// TIA Portal V17 export
// export: Created 2025-08-05T09:36:01.5993523Z, ExportSetting WithDefaults, DisplayName Totally Integrated Automation Portal, DisplayVersion V17, DisplayName TIA Portal Openness, DisplayVersion V17, DisplayName TIA Portal Version Control Interface, DisplayVersion V17, DisplayName SINAMICS Startdrive Advanced, DisplayVersion V17, DisplayName SINAMICS Startdrive G130, G150, S120, S150, SINAMICS MV, S210, DisplayVersion V17, DisplayName SINAMICS Startdrive G110M, G120, G120C, G120D, G120P, G115D, DisplayVersion V17, DisplayName STEP 7 Professional, DisplayVersion V17, DisplayName STEP 7 Safety, DisplayVersion V17, DisplayName WinCC Advanced, DisplayVersion V17
TYPE "API_Outputs"
// stored: IsFailsafeCompliant false
   STRUCT
      Job_Comp_Ack : Bool;   // Acknowledge the Job Complete Signal has been Received
      Tx : DInt;   // Transmission Counter
      Job : DInt;   // Middleware Job Command
      Serial_Number : Array[1..32] of Char;   // Serial Number of Part to Be Loaded to LDD File
      Part_Type : Array[1..18] of Char;   // Part Type in Station
      LDD : Struct   // Laser Depth Dynamics
         Sequence_Mask : Array[0.."LASERCOMM_LDD_ARRAY_SIZE"] of Bool;   // Weld Mask for Skipping Welds in an LDD Sequence
      END_STRUCT;
   END_STRUCT;
END_TYPE
